// TIA Portal project "Alternancia-De-Bombas" (V18)

(* hardware
DEVICE "S7-1200 station_1"  S7-1200 Station
   slot 0: "Rack_0"  S7-1200 Rack  Rack  V1.0
   slot 1: "PLC_1"  CPU 1214C DC/DC/Rly  6ES7 214-1HG40-0XB0  V4.4
*)

// ===== PLC "PLC_1"  CPU 1214C DC/DC/Rly =====

VAR_GLOBAL   // PLC tag table "Default tag table"
   "System_Byte" AT %MB1 : Byte;
   "FirstScan" AT %M1.0 : Bool;
   "DiagStatusUpdate" AT %M1.1 : Bool;
   "AlwaysTRUE" AT %M1.2 : Bool;
   "AlwaysFALSE" AT %M1.3 : Bool;
   "Clock_Byte" AT %MB0 : Byte;
   "Clock_10Hz" AT %M0.0 : Bool;
   "Clock_5Hz" AT %M0.1 : Bool;
   "Clock_2.5Hz" AT %M0.2 : Bool;
   "Clock_2Hz" AT %M0.3 : Bool;
   "Clock_1.25Hz" AT %M0.4 : Bool;
   "Clock_1Hz" AT %M0.5 : Bool;
   "Clock_0.625Hz" AT %M0.6 : Bool;
   "Clock_0.5Hz" AT %M0.7 : Bool;
   "Tag_1" AT %MD500 : Real;
   "Tag_2" AT %MD501 : Real;
END_VAR

VAR_GLOBAL   // PLC tag table "Entras-Salidas"
   "KMbomba1" AT %Q0.0 : Bool;
   "KMbomba2" AT %Q0.2 : Bool;
   "luzFalla" AT %Q0.1 : Bool;
   "Reset" AT %I0.1 : Bool;
   "Presion" AT %IW64 : Int;
   "Temp" AT %IW66 : Int;
   "SalidaTemp" AT %MD100 : DWord;
   "SalidaPresion" AT %MD101 : DWord;
   "IntTemp" AT %MD201 : DWord;
   "IntPresion" AT %MD202 : DWord;
   "Auto-Manual" AT %M2.1 : Bool;
END_VAR

VAR_GLOBAL   // PLC tag table "Tag table_1"
   "Mbomba1" AT %M2.4 : Bool;
   "Mbomba2" AT %M2.5 : Bool;
   "LuzFallaPresion" AT %M2.6 : Bool;
   "LuzFallaTemp" AT %M2.7 : Bool;
END_VAR

DATA_BLOCK "PLC"   // DB1
{ S7_Optimized_Access := 'TRUE' }
VERSION : 0.1
   VAR
      "Act.LuzFalla" : Bool;
      "Act.Bomba1" : Bool;
      "Act.Bomba2" : Bool;
      FallaPresion : Bool;
      FallaTemperatura : Bool;
      FallaCritica : Bool;
   END_VAR
BEGIN
END_DATA_BLOCK

FUNCTION "Salidas" : Void   // FC1, SCL
{ S7_Optimized_Access := 'TRUE' }
VERSION : 0.1
BEGIN
   "luzFalla" := "PLC"."Act.LuzFalla" AND "Clock_1Hz";
   "KMbomba1" := "PLC"."Act.Bomba1";
   "KMbomba2" := "PLC"."Act.Bomba2";
END_FUNCTION

ORGANIZATION_BLOCK "AnalogInputs"   // OB1, LAD, ProgramCycle
TITLE = "Main Program Sweep (Cycle)"
{ S7_Optimized_Access := 'TRUE' }
VERSION : 0.1
   VAR_INPUT
      Initial_Call : Bool;   // Initial call of this OB
      Remanence : Bool;   // =True, if remanent data are available
   END_VAR
BEGIN

REGION Network 1
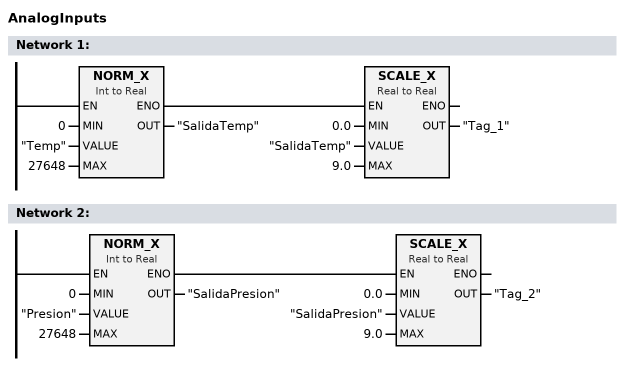
   RUNG wire#powerrail
      { S7_Templates := "[SrcType := Int, DestType := Real]" } Normalize(min := 0, value := "Temp", max := 27648, out => "SalidaTemp")
      { S7_Templates := "[SrcType := Real, DestType := Real]" } Scale(min := 0.0, value := "SalidaTemp", max := 9.0, out => "Tag_1")
   END_RUNG
   // the same network as SCL:
   "SalidaTemp" := NORM_X(MIN := 0, VALUE := "Temp", MAX := 27648);
   "Tag_1" := SCALE_X(MIN := 0.0, VALUE := "SalidaTemp", MAX := 9.0);
END_REGION

REGION Network 2
   RUNG wire#powerrail
      { S7_Templates := "[SrcType := Int, DestType := Real]" } Normalize(min := 0, value := "Presion", max := 27648, out => "SalidaPresion")
      { S7_Templates := "[SrcType := Real, DestType := Real]" } Scale(min := 0.0, value := "SalidaPresion", max := 9.0, out => "Tag_2")
   END_RUNG
   // the same network as SCL:
   "SalidaPresion" := NORM_X(MIN := 0, VALUE := "Presion", MAX := 27648);
   "Tag_2" := SCALE_X(MIN := 0.0, VALUE := "SalidaPresion", MAX := 9.0);
END_REGION
END_ORGANIZATION_BLOCK

ORGANIZATION_BLOCK "LogicaScl"   // OB123, SCL, ProgramCycle
TITLE = "Main Program Sweep (Cycle)"
{ S7_Optimized_Access := 'TRUE' }
VERSION : 0.1
   VAR_INPUT
      Initial_Call : Bool;   // Initial call of this OB
      Remanence : Bool;   // =True, if remanent data are available
   END_VAR
BEGIN
   "Salidas"();
   IF NOT "Auto-Manual" THEN
       IF NOT "PLC".FallaCritica AND "Mbomba2" THEN
           "PLC"."Act.Bomba2" := TRUE;
           "PLC"."Act.Bomba1" := FALSE;
       ELSIF NOT "PLC".FallaCritica AND "Mbomba1" THEN
             "PLC"."Act.Bomba1" := TRUE;
             "PLC"."Act.Bomba2" := FALSE;
         ELSIF "PLC".FallaCritica THEN
             "PLC"."Act.Bomba1" := FALSE;
             "PLC"."Act.Bomba2" := FALSE;
         END_IF;
    END_IF;
END_ORGANIZATION_BLOCK

ORGANIZATION_BLOCK "ActivacionDeFallas"   // OB124, SCL, ProgramCycle
TITLE = "Main Program Sweep (Cycle)"
{ S7_Optimized_Access := 'TRUE' }
VERSION : 0.1
   VAR_INPUT
      Initial_Call : Bool;   // Initial call of this OB
      Remanence : Bool;   // =True, if remanent data are available
   END_VAR
BEGIN
   "PLC"."Act.LuzFalla" := "Tag_1" < 6 AND "Tag_2" > 6;
END_ORGANIZATION_BLOCK